// TIA Portal project "robot_5_dof" (V15)

(* hardware
DEVICE "GSD device_1"  GSD.Device.PN
   slot 0: "Rack"  Rack  V1.0
   slot 0: "al1100"  AL1100  AL1100
      slot 0: "AL1100"  AL1100
      slot 1: "4 Ports_1"  4 Ports  AL1100
         slot 0: "IO-Link Master"  IO-Link Master
      slot 1: "X1"  X1
         slot 1: "Port 1"  Port 1
         slot 2: "Port 2"  Port 2
   slot 1: "IO-Link In  2 Byte + PQI"  IO-Link In  2 Byte + PQI
   slot 2: "Disabled"  Disabled
   slot 3: "IO-Link In  2 Byte + PQI_1"  IO-Link In  2 Byte + PQI
   slot 4: "Disabled_1"  Disabled
DEVICE "S7-1200 station_1"  S7-1200 Station
   slot 0: "Rack_0"  S7-1200 Rack  Rack  V1.0
   slot 1: "PLC_1"  CPU 1215C DC/DC/DC  6ES7 215-1AG40-0XB0  V4.2
      slot 3: "AQ 1x12BIT_1"  AQ1 signal board  6ES7 232-4HA30-0XB0  V1.0
   slot 2: "DI 16/DQ 16x24VDC_1"  6ES7 223-1BL32-0XB0  V2.0
   slot 101: "CM 1241 (RS232)_1"  6ES7 241-1AH30-0XB0  V1.0
*)

// ===== PLC "PLC_1"  CPU 1215C DC/DC/DC =====

VAR_GLOBAL   // PLC tag table "Default tag table"
   "Tag_1" AT %IW68 : UInt;
   "end_sensor" AT %IW75 : UInt;
   "Tag_3" AT %IW71 : UInt;
   "start_sensor" AT %IW80 : UInt;
   "System_Byte" AT %MB1 : Byte;
   "FirstScan" AT %M1.0 : Bool;
   "DiagStatusUpdate" AT %M1.1 : Bool;
   "AlwaysTRUE" AT %M1.2 : Bool;
   "AlwaysFALSE" AT %M1.3 : Bool;
   "Clock_Byte" AT %MB0 : Byte;
   "Clock_10Hz" AT %M0.0 : Bool;
   "Clock_5Hz" AT %M0.1 : Bool;
   "Clock_2.5Hz" AT %M0.2 : Bool;
   "Clock_2Hz" AT %M0.3 : Bool;
   "Clock_1.25Hz" AT %M0.4 : Bool;
   "Clock_1Hz" AT %M0.5 : Bool;
   "Clock_0.625Hz" AT %M0.6 : Bool;
   "Clock_0.5Hz" AT %M0.7 : Bool;
   "Tag_5" AT %MB10 : Byte;
   "Tag_6" AT %MW12 : Word;
   "Tag_7" AT %MW14 : Word;
   "Tag_8" AT %M10.0 : Bool;
   "Tag_9" AT %M11.0 : Bool;
   "send_cmd" AT %M15.0 : Bool;
   "K1" AT %M20.0 : Bool;
   "K2" AT %M21.0 : Bool;
   "K3" AT %M22.0 : Bool;
   "K4" AT %M23.0 : Bool;
   "K5" AT %M24.0 : Bool;
   "K6" AT %M25.0 : Bool;
   "K7" AT %M26.0 : Bool;
   "K8" AT %M27.0 : Bool;
   "Tag_2" AT %I0.6 : Bool;
   "Tag_4" AT %I8.0 : Bool;
   "Start Button" AT %I8.6 : Bool;
   "System_Byte(1)" AT %MB1 : Byte;
   "Tag_10" AT %Q0.7 : Bool;
   "conveyor" AT %Q8.7 : Bool;
   "reset_buffer" AT %M30.0 : Bool;
   "Tag_11" AT %M40.0 : Bool;
END_VAR

DATA_BLOCK "Data_block_2"   // DB4
{ S7_Optimized_Access := 'TRUE' }
VERSION : 0.1
   VAR
      Rx : Array[0..3] of Byte;
   END_VAR
BEGIN
   Rx[0] := 0;
   Rx[1] := 0;
   Rx[2] := 0;
   Rx[3] := 0;
END_DATA_BLOCK

DATA_BLOCK "Data_block_1"   // DB5
{ S7_Optimized_Access := 'TRUE' }
VERSION : 0.1
   VAR
      DATA : Array[0..3] of Byte;
   END_VAR
BEGIN
   DATA[0] := 0;
   DATA[1] := 0;
   DATA[2] := 0;
   DATA[3] := 0;
END_DATA_BLOCK

DATA_BLOCK "State"   // DB7
{ S7_Optimized_Access := 'TRUE' }
VERSION : 0.1
   VAR
      State : DInt;
   END_VAR
BEGIN
END_DATA_BLOCK

ORGANIZATION_BLOCK "Main"   // OB1, LAD, ProgramCycle
TITLE = "Main Program Sweep (Cycle)"
{ S7_Optimized_Access := 'TRUE' }
VERSION : 0.1
   VAR_INPUT
      Initial_Call : Bool;   // Initial call of this OB
      Remanence : Bool;   // =True, if remanent data are available
   END_VAR
   VAR_TEMP   // added for the SCL form of the ladder/FBD networks
      _w1 : Bool;
   END_VAR
BEGIN

REGION Network 1
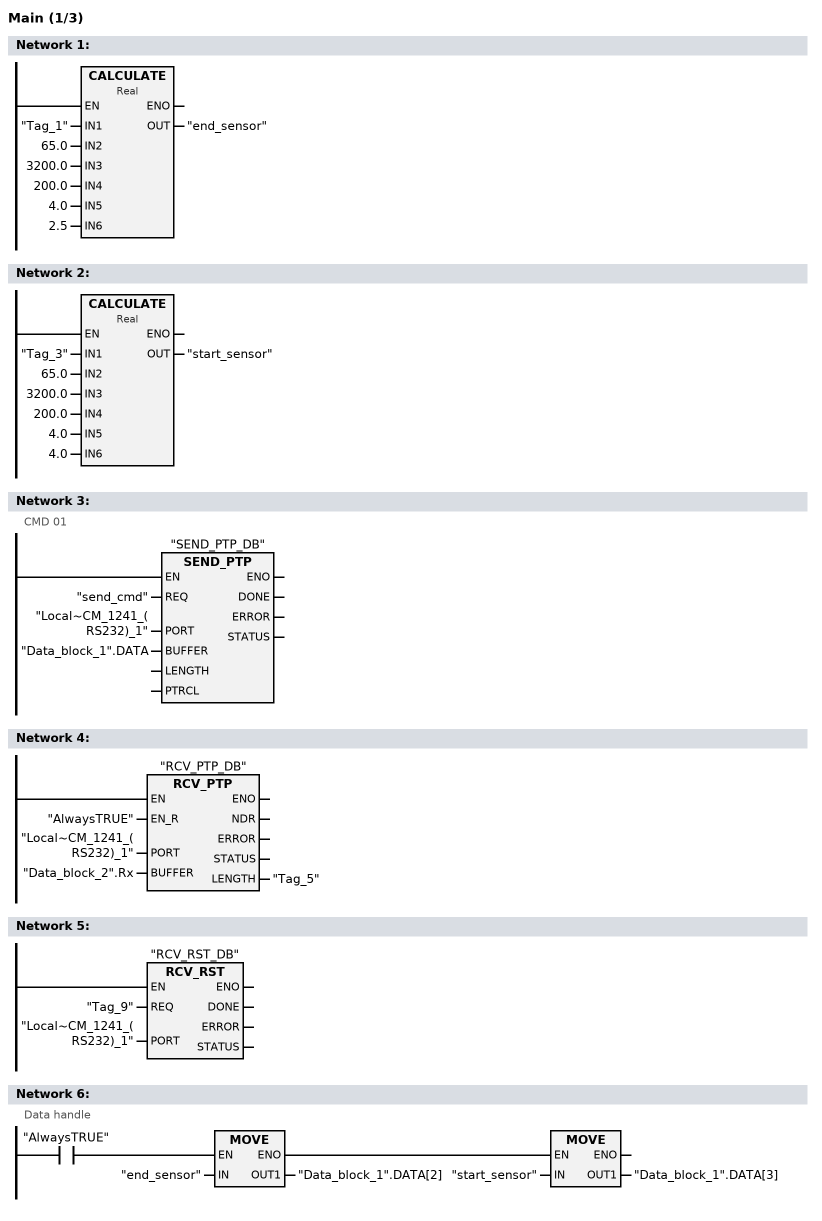
   RUNG wire#powerrail
      { S7_Templates := "SrcType := Real"; S7_GenerateENO := "TRUE"; S7_Expression := "(((IN4-IN5)/(IN3-IN2))*(IN1-IN2))+IN5-IN6" } Calculate(in1 := "Tag_1", in2 := 65.0, in3 := 3200.0, in4 := 200.0, in5 := 4.0, in6 := 2.5, out => "end_sensor")
   END_RUNG
   // the same network as SCL:
   "end_sensor" := (((200.0-4.0)/(3200.0-65.0))*("Tag_1"-65.0))+4.0-2.5;
END_REGION

REGION Network 2
   RUNG wire#powerrail
      { S7_Templates := "SrcType := Real"; S7_GenerateENO := "TRUE"; S7_Expression := "(((IN4-IN5)/(IN3-IN2))*(IN1-IN2))+IN5-IN6" } Calculate(in1 := "Tag_3", in2 := 65.0, in3 := 3200.0, in4 := 200.0, in5 := 4.0, in6 := 4.0, out => "start_sensor")
   END_RUNG
   // the same network as SCL:
   "start_sensor" := (((200.0-4.0)/(3200.0-65.0))*("Tag_3"-65.0))+4.0-4.0;
END_REGION

REGION Network 3
   // CMD 01
   "SEND_PTP_DB"(REQ := "send_cmd", PORT := "Local~CM_1241_(RS232)_1", BUFFER := "Data_block_1".DATA);   // SEND_PTP
END_REGION

REGION Network 4
   "RCV_PTP_DB"(EN_R := "AlwaysTRUE",   // RCV_PTP
                PORT := "Local~CM_1241_(RS232)_1",
                BUFFER := "Data_block_2".Rx,
                LENGTH => "Tag_5");
END_REGION

REGION Network 5
   "RCV_RST_DB"(REQ := "Tag_9", PORT := "Local~CM_1241_(RS232)_1");   // RCV_RST
END_REGION

REGION Network 6
   // Data handle
   RUNG wire#powerrail
      Contact( "AlwaysTRUE" )
      { S7_GenerateENO := "TRUE" } Move(in := "end_sensor", out1 => "Data_block_1".DATA[2])
      { S7_GenerateENO := "TRUE" } Move(in := "start_sensor", out1 => "Data_block_1".DATA[3])
   END_RUNG
   // the same network as SCL:
   // ENO of a box is taken as its EN; it also drops when the box reports an error
   IF "AlwaysTRUE" THEN
       "Data_block_1".DATA[2] := "end_sensor";
       "Data_block_1".DATA[3] := "start_sensor";
   END_IF;
END_REGION

REGION Network 7
   // State machine
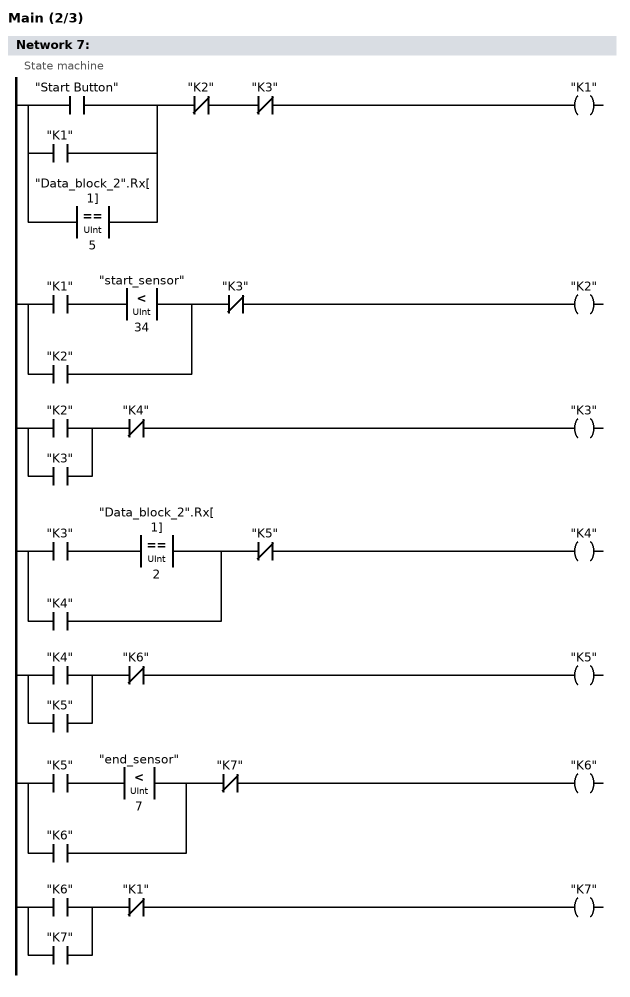
   RUNG wire#powerrail
      Contact( "Start Button" )
      wire#w1
      I_Contact( "K2" )
      I_Contact( "K3" )
      Coil( "K1" )
   END_RUNG
   RUNG wire#powerrail
      Contact( "K1" )
   END_RUNG wire#w1
   RUNG wire#powerrail
      { S7_Templates := "SrcType := UInt" } EQ_Contact(in1 := "Data_block_2".Rx[1], in2 := 5)
   END_RUNG wire#w1
   RUNG wire#powerrail
      Contact( "K1" )
      { S7_Templates := "SrcType := UInt" } LT_Contact(in1 := "start_sensor", in2 := 34)
      wire#w2
      I_Contact( "K3" )
      Coil( "K2" )
   END_RUNG
   RUNG wire#powerrail
      Contact( "K2" )
   END_RUNG wire#w2
   RUNG wire#powerrail
      Contact( "K2" )
      wire#w3
      I_Contact( "K4" )
      Coil( "K3" )
   END_RUNG
   RUNG wire#powerrail
      Contact( "K3" )
   END_RUNG wire#w3
   RUNG wire#powerrail
      Contact( "K3" )
      { S7_Templates := "SrcType := UInt" } EQ_Contact(in1 := "Data_block_2".Rx[1], in2 := 2)
      wire#w4
      I_Contact( "K5" )
      Coil( "K4" )
   END_RUNG
   RUNG wire#powerrail
      Contact( "K4" )
   END_RUNG wire#w4
   RUNG wire#powerrail
      Contact( "K4" )
      wire#w5
      I_Contact( "K6" )
      Coil( "K5" )
   END_RUNG
   RUNG wire#powerrail
      Contact( "K5" )
   END_RUNG wire#w5
   RUNG wire#powerrail
      Contact( "K5" )
      { S7_Templates := "SrcType := UInt" } LT_Contact(in1 := "end_sensor", in2 := 7)
      wire#w6
      I_Contact( "K7" )
      Coil( "K6" )
   END_RUNG
   RUNG wire#powerrail
      Contact( "K6" )
   END_RUNG wire#w6
   RUNG wire#powerrail
      Contact( "K6" )
      wire#w7
      I_Contact( "K1" )
      Coil( "K7" )
   END_RUNG
   RUNG wire#powerrail
      Contact( "K7" )
   END_RUNG wire#w7
   // the same network as SCL:
   "K1" := ("Start Button" OR "K1" OR ("Data_block_2".Rx[1] = 5)) AND NOT "K2" AND NOT "K3";
   "K2" := (("K1" AND ("start_sensor" < 34)) OR "K2") AND NOT "K3";
   "K3" := ("K2" OR "K3") AND NOT "K4";
   "K4" := (("K3" AND ("Data_block_2".Rx[1] = 2)) OR "K4") AND NOT "K5";
   "K5" := ("K4" OR "K5") AND NOT "K6";
   "K6" := (("K5" AND ("end_sensor" < 7)) OR "K6") AND NOT "K7";
   "K7" := ("K6" OR "K7") AND NOT "K1";
END_REGION

REGION Network 8
   // State control
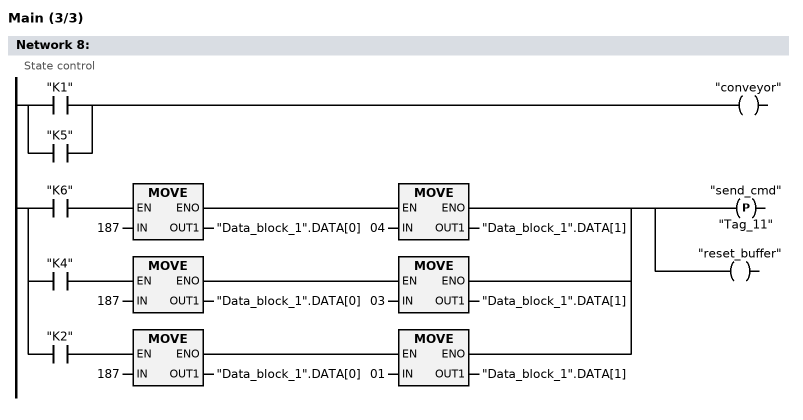
   // ENO of a box is taken as its EN; it also drops when the box reports an error
   "conveyor" := "K1" OR "K5";
   IF "K6" THEN
       "Data_block_1".DATA[0] := 187;
       "Data_block_1".DATA[1] := 04;
   END_IF;
   IF "K4" THEN
       "Data_block_1".DATA[0] := 187;
       "Data_block_1".DATA[1] := 03;
   END_IF;
   IF "K2" THEN
       "Data_block_1".DATA[0] := 187;
       "Data_block_1".DATA[1] := 01;
   END_IF;
   #_w1 := "K6" OR "K4" OR "K2";
   "send_cmd" := #_w1 AND NOT "Tag_11";   // rising edge
   "Tag_11" := #_w1;
   "reset_buffer" := #_w1;
END_REGION
END_ORGANIZATION_BLOCK